// TIA Portal project "encoder_giris" (V18)

(* hardware
DEVICE "S7-1200 station_1"  S7-1200 Station
   slot 0: "Rack_0"  S7-1200 Rack  Rack  V1.0
   slot 1: "PLC_1"  CPU 1214C DC/DC/DC  6ES7 214-1AG40-0XB0  V4.6
*)

// ===== PLC "PLC_1"  CPU 1214C DC/DC/DC =====

VAR_GLOBAL   // PLC tag table "Default tag table"
   "İLERİ START" AT %M0.0 : Bool;
   "ÇIKIŞ 0" AT %Q0.0 : Bool;
   "GERİ START" AT %M0.1 : Bool;
   "ÇIKIŞ 1" AT %Q0.1 : Bool;
   "SABİT HIZ 1" AT %M0.2 : Bool;
   "ÇIKIŞ 2" AT %Q0.2 : Bool;
   "SABİT HIZ 2" AT %M0.3 : Bool;
   "ÇIKIŞ 3" AT %Q0.3 : Bool;
   "Tag_1" AT %M20.0 : Bool;
   "Tag_2" AT %MD60 : DWord;
   "Tag_3" AT %MW90 : Word;
   "Tag_4" AT %QW80 : Word;
   "HSC5 ADRESI" AT %ID1016 : DWord;
   "HSC5_ATAMA" AT %MD30 : DWord;
END_VAR

ORGANIZATION_BLOCK "Main"   // OB1, LAD, ProgramCycle
TITLE = "Main Program Sweep (Cycle)"
{ S7_Optimized_Access := 'TRUE' }
VERSION : 0.1
// Device view kısmından kaç tane HSC var görebiliyoruz
// Properties kısmından ise HSCleri kontrol edebiliyoruz
   VAR_INPUT
      Initial_Call : Bool;   // Initial call of this OB
      Remanence : Bool;   // =True, if remanent data are available
   END_VAR
BEGIN

REGION Network 1
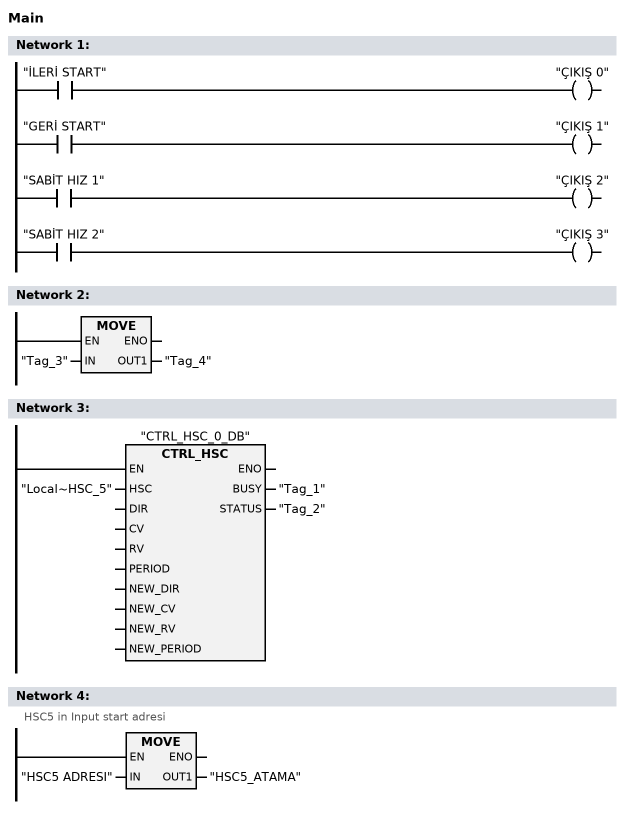
   RUNG wire#powerrail
      Contact( "İLERİ START" )
      Coil( "ÇIKIŞ 0" )
   END_RUNG
   RUNG wire#powerrail
      Contact( "GERİ START" )
      Coil( "ÇIKIŞ 1" )
   END_RUNG
   RUNG wire#powerrail
      Contact( "SABİT HIZ 1" )
      Coil( "ÇIKIŞ 2" )
   END_RUNG
   RUNG wire#powerrail
      Contact( "SABİT HIZ 2" )
      Coil( "ÇIKIŞ 3" )
   END_RUNG
   // the same network as SCL:
   "ÇIKIŞ 0" := "İLERİ START";
   "ÇIKIŞ 1" := "GERİ START";
   "ÇIKIŞ 2" := "SABİT HIZ 1";
   "ÇIKIŞ 3" := "SABİT HIZ 2";
END_REGION

REGION Network 2
   RUNG wire#powerrail
      Move(in := "Tag_3", out1 => "Tag_4")
   END_RUNG
   // the same network as SCL:
   "Tag_4" := "Tag_3";
END_REGION

REGION Network 3
   "CTRL_HSC_0_DB"(HSC := "Local~HSC_5", BUSY => "Tag_1", STATUS => "Tag_2");   // CTRL_HSC
END_REGION

REGION Network 4
   // HSC5 in Input start adresi
   RUNG wire#powerrail
      Move(in := "HSC5 ADRESI", out1 => "HSC5_ATAMA")
   END_RUNG
   // the same network as SCL:
   "HSC5_ATAMA" := "HSC5 ADRESI";
END_REGION
END_ORGANIZATION_BLOCK